TYPE ST_ControlStewart :
STRUCT
	eta : ARRAY [0..5] OF LREAL;
END_STRUCT
END_TYPE

(* stored: Version 1.1.0.1, ProductVersion 3.1.4022.7
   DUT ST_ControlStewart: Id {f6680c9a-ba32-4cdf-b6e9-dd2896846b77} *)
